RoboDK station: Simulation_roboDK.rdk

Station Simulation_roboDK (saved by RoboDK 5.7.3). Poses are relative to the parent item; angles as X-Y-Z fixed-axis rotations.
  - object Manikin_1 at (0, 0, 0) mm, geometry from Manikin_1.STEP
  - frame Human_Base at (0, 958, 0) mm
    - frame hipL_abduction at (63.26, -78.51, -37.42) mm, rotated rx 0 ry 0 rz -7.94 deg
      - frame hipL_flexion at (0, 0, 0) mm
        - frame hipL_rotation at (0, 0, 0) mm
          - frame kneeL_flexion at (67.44, -393.44, -12.97) mm
            - frame ankleL_flexion at (42.46, -394.54, 0) mm, rotated rx 0 ry 0 rz 7.94 deg
              - item type 7 Manikin_1-pied_g
            - item type 7 Manikin_1-tibia_g
          - item type 7 Manikin_1-cuisse_g
    - frame shoulderL_abduction at (206.4, 423.68, 12.96) mm, rotated rx 0 ry 0 rz -42 deg
      - frame shoulderL_flexion at (0, 0, 0) mm
        - frame shoulderL_rotation at (0, 0, 0) mm
          - frame elbowL_flexion at (155.8, -191.9, 27.9) mm
            - frame wristL_flexion at (148.7, -146.81, 80.89) mm
              - frame wristL_deviation at (0, 0, 0) mm
                - item type 7 Manikin_1-main_g
            - item type 7 Manikin_1-avant_bras_g
          - item type 7 Manikin_1-bras_g
    - frame hipR_abduction at (-70.11, -75.34, -37.06) mm, rotated rx 0 ry 0 rz 10.84 deg
      - frame hipR_flexion at (0, 0, 0) mm
        - frame hipR_rotation at (0, 0, 0) mm
          - frame kneeR_flexion at (-86.5, -385.51, -37.91) mm
            - frame ankleR_flexion at (-60.5, -382.31, -26.03) mm, rotated rx 0 ry 0 rz -10.84 deg
              - item type 7 Manikin_1-pied_d_1
              - item type 7 Manikin_1-pied_d_2
            - item type 7 Manikin_1-tibia_d_1
            - item type 7 Manikin_1-tibia_d_2
          - item type 7 Manikin_1-cuisse_d
    - frame shoulderR_abduction at (-136.98, 400.49, -20) mm, rotated rx 0 ry 0 rz -63.21 deg
      - frame shoulderR_flexion at (0, 0, 0) mm, rotated rx 57.65 ry 0 rz 0 deg
        - frame shoulderR_rotation at (0, 0, 0) mm, rotated rx 0 ry 29.61 rz 0 deg
          - frame elbowR_flexion at (-80.76, -228.86, 52.14) mm, rotated rx -95.28 ry 0 rz 0 deg
            - frame forearmR_rotation at (0, 0, 0) mm, rotated rx 0 ry 25.7 rz 0 deg
              - frame wristR_flexion at (-76.34, -195.54, 87.27) mm, rotated rx -9.18 ry 0 rz 0 deg
                - frame wristR_deviation at (0, 0, 0) mm, rotated rx 0 ry 0 rz 5.97 deg
                  - item type 7 Manikin_1-main_d
              - item type 7 Manikin_1-avant_bras_d
          - item type 7 Manikin_1-bras_d
    - item type 7 Manikin_1-bassin
    - item type 7 Manikin_1-tete
    - item type 7 Manikin_1-torso
  - Python program fix_segments (listed below)
  - object Table at (0, 900, 485) mm, size 1100 x 900 x 550 mm
  - object Piece at (80, 940, 300) mm, size 80 x 80 x 80 mm
  - Python program play_trajectory_robodk (listed below)
  - Python program Position_0 (listed below)

--- Python program fix_segments ---
# -*- coding: utf-8 -*-
"""
fix_reattache_segments.py — Repare le mannequin eclate a la reouverture du
.rdk SANS rebuild (quelques secondes), en re-jouant le re-basage geometrique
perdu a la sauvegarde.

Cause (diagnostic du 10/06) : pour les sous-solides type 7 (courbes issues
du Split), le .rdk sauve les points BRUTS d'origine — la compensation posee
par setParentStatic au moment du rig n'est PAS persistee. A l'ouverture,
RoboDK applique la transformation du frame parent sur ces points bruts
-> double transformation -> mannequin eclate. Les frames, vrais items a
pose persistee, restent corrects.

Remede, segment par segment :
  1) memoriser la pose relative de chaque frame, puis remettre chaque
     frame en etat de CONSTRUCTION (translation seule, rotation identite —
     l'etat dans lequel le rig d'origine a pose ses compensations)
  2) setParent(station)      — detache en KEEP-RELATIVE : la compensation
     (identite au chargement) ne change pas -> le segment retombe sur ses
     points bruts = position d'import, mannequin recompose
     setParentStatic(frame)  — re-attache en preservant l'absolu : la
     compensation F_build^-1 est re-posee, exactement comme au rig
  3) restaurer les poses memorisees (garde-a-vous, jambes resserrees) :
     la geometrie suit les frames

!! NE PAS envelopper dans RDK.Render(False) : le re-basage des type 7
echoue silencieusement sans rendu actif (constate le 10/06 — deux
tentatives identiques en Render(False) = aucun effet, la meme sequence
render actif fonctionne).

A relancer A CHAQUE OUVERTURE du .rdk (la sauvegarde re-perd le re-basage).
Filet de securite si etat incoherent : scripts/rebuild_operateur.py (~30 s).

!! PAS IDEMPOTENT : sur une station SAINE (fraichement rebuildee ou deja
reparee), le re-basage s'appliquerait une fois de trop et eclaterait le
mannequin. Une garde detecte l'etat via un segment du tronc et refuse de
tourner si la station est saine (--force pour outrepasser).

Usage (RoboDK ouvert, station chargee) :
    python fix_reattache_segments.py [--skip nom1,nom2] [--force]
    --skip  : segments a ne pas toucher (ex. deja repares a la main)
    --force : sauter la garde de detection
"""
import math
import sys
import time
from pathlib import Path
sys.path.insert(0, str(Path(__file__).resolve().parent))
from robolink import Robolink, ITEM_TYPE_FRAME
from robodk.robomath import transl

# ancres d'import des segments du tronc (cf. build_human_robodk.ANCHORS),
# en dur pour que le script reste autonome une fois embarque dans la station
TRONC = {"tete": (20, 1584, 30), "torso": (15, 1260, 0), "bassin": (0, 958, 0)}

skip = set()
if "--skip" in sys.argv:
    skip = set(sys.argv[sys.argv.index("--skip") + 1].split(","))

t0 = time.time()
RDK = Robolink()
station = RDK.ActiveStation()
print("Station :", station.Name())


def _d(a, b):
    return math.sqrt(sum((x - y) ** 2 for x, y in zip(a, b)))


def garde_station_cassee():
    """True si le mannequin est eclate (double transformation detectee)."""
    for it in RDK.ItemList():
        if it.Type() != 7:
            continue
        part = it.Name().split("-", 1)[-1]
        if part not in TRONC:
            continue
        bb = it.setParam("BoundingBox")
        c = [(bb["min"][i] + bb["max"][i]) / 2.0 for i in range(3)]
        a = TRONC[part]
        F = it.Parent().PoseAbs().rows
        fa = [sum(F[i][j] * a[j] for j in range(3)) + F[i][3] for i in range(3)]
        d_sain, d_casse = _d(c, a), _d(c, fa)
        etat = "CASSEE (double transformation)" if d_casse < d_sain else "saine"
        print(f"Garde ({part}) : d_sain={d_sain:.0f} mm, d_casse={d_casse:.0f} mm -> station {etat}")
        return d_casse < d_sain
    sys.exit("Garde impossible : aucun segment du tronc (tete/torso/bassin) trouve.")


if "--force" not in sys.argv and not garde_station_cassee():
    sys.exit("Rien a faire — relancer avec --force pour outrepasser la garde.")

frames = RDK.ItemList(ITEM_TYPE_FRAME)
solids = [it for it in RDK.ItemList() if it.Type() == 7]
if not solids:
    sys.exit("Rien a reparer : aucun sous-solide type 7 dans la station.")
parent_of = {}
for s in solids:
    nm = s.Name()
    if nm in skip or nm.split("-", 1)[-1] in skip:
        print(f"  (skip : {nm})")
        continue
    p = s.Parent()
    if p.Type() == 3:
        parent_of[s] = p
    else:
        print(f"  (ignore : {nm} n'est pas sous un frame)")
print(f"{len(frames)} frames, {len(parent_of)} segments a re-attacher")

# 1) frames -> etat de construction (translation seule)
saved = []
for fr in frames:
    pose = fr.Pose()
    saved.append((fr, pose))
    r = pose.rows
    fr.setPose(transl(r[0][3], r[1][3], r[2][3]))

# 2) re-basage : detacher en keep-relative, re-attacher en statique
for s, fr in parent_of.items():
    s.setParent(station)
    s.setParentStatic(fr)
    print(f"  re-attache : {s.Name():26s} -> {fr.Name()}")

# 3) restaurer les poses (garde-a-vous, jambes resserrees, ...)
for fr, pose in saved:
    fr.setPose(pose)

print(f"OK — {len(parent_of)} segments re-attaches en {time.time() - t0:.1f} s")

--- Python program play_trajectory_robodk ---
# -*- coding: utf-8 -*-
"""
play_trajectory_robodk.py

Plays back a precomputed 7-DOF joint trajectory (from
src/export_trajectory_for_robodk.py) on a RoboDK mannequin arm -- the
playback half of the PINN/RoboDK digital-twin integration (see chat,
2026-08-10). Deliberately mirrors old/Tache_Bras.py's own structure
(Robolink() + named Frame items + REST pose * local rotation + fixed-rate
render loop) since that's the established, working pattern in this
project for animating this kind of rig -- just without Tache_Bras's IK/
choreography, since here the trajectory is already fully precomputed by
the PINN.

Run this under RoboDK's OWN embedded Python (has robodk/robolink/numpy
already, confirmed 2026-08-10), with the target RoboDK station open:
    C:\\RoboDK\\Python-Embedded\\python.exe play_trajectory_robodk.py <csv_path>

IMPORTANT -- JOINT_MAP below is an unverified best guess and WILL need
your input once the new 7-DOF station exists:
  - rig_frame: must match the exact Frame item name in your new station.
    Left blank (None) for all 7 by default -- fill these in first, the
    script exits immediately listing what it can't find otherwise.
  - axis: which local axis (x/y/z) that frame rotates about. Copied from
    old/config.py's SEGMENTS (the existing 7-DOF chain scaffold in this
    project) as a starting point -- verify against however you actually
    build the new joints, they may not match.
  - sign: +1 or -1. DBAS22's angle convention for a given column is not
    guaranteed to match whichever direction you wire the corresponding
    RoboDK axis to rotate. Use --probe (below) to check each joint
    in isolation and flip signs until the motion looks anatomically
    correct, exactly how Tache_Bras.py's original author calibrated
    elbowL_flexion's sign via manual probing (see its "_probe_coude"
    comment) -- there's no way to get this right without the actual rig
    in front of you.

Usage:
    play_trajectory_robodk.py <csv_path>              play back a trajectory
    play_trajectory_robodk.py --probe [step_deg]       one joint at a time,
                                                        +step_deg (default 20)
                                                        from rest, paused for
                                                        visual check between
                                                        each -- run this FIRST
"""
import csv
import math
import sys
from pathlib import Path

from robolink import Robolink, ITEM_TYPE_FRAME
from robodk.robomath import rotx, roty, rotz

# DBAS22 column -> (rig frame name, local axis, sign). Order matches
# dataset.JOINT_COLS (sp, sr, ay, ep, fy, hp, hr); rig frame names/axes
# follow old/config.py's SEGMENTS naming (shoulder_abduction, ...,
# wrist_deviation) as a starting point -- see module docstring.
JOINT_MAP = {
    # Frame names confirmed against the live station (Simulation_roboDK.rdk,
    # 2026-08-10) via robolink -- RIGHT arm, since s1 (the trial used in
    # trajectories/s1_tgt50_*.csv) is right-handed (arm_side='R'). Axes/
    # signs are still the config.py-derived best guess -- run --probe
    # before trusting them.
    "sp": {"rig_frame": "shoulderR_flexion", "axis": "x", "sign": +1},
    "sr": {"rig_frame": "shoulderR_abduction", "axis": "z", "sign": +1},
    "ay": {"rig_frame": "shoulderR_rotation", "axis": "y", "sign": +1},
    "ep": {"rig_frame": "elbowR_flexion", "axis": "x", "sign": +1},
    "fy": {"rig_frame": "forearmR_rotation", "axis": "y", "sign": +1},
    "hp": {"rig_frame": "wristR_flexion", "axis": "x", "sign": +1},
    "hr": {"rig_frame": "wristR_deviation", "axis": "z", "sign": +1},
}
ROT = {"x": rotx, "y": roty, "z": rotz}

DT = 0.04  # s/frame during playback (~25 fps of applied poses; actual
           # wall-clock rate is capped by RoboDK's render time, same
           # caveat Tache_Bras.py notes for its own DT)


def _load_csv(path):
    with open(path, newline="") as f:
        r = csv.reader(f)
        header = next(r)
        rows = [[float(x) for x in row] for row in r]
    cols = {name: i for i, name in enumerate(header)}
    return header, cols, rows


def _get_frames(rdk):
    frames = {}
    missing = []
    for col, spec in JOINT_MAP.items():
        name = spec["rig_frame"]
        if name is None:
            missing.append(f"{col} (rig_frame not set)")
            continue
        fr = rdk.Item(name, ITEM_TYPE_FRAME)
        if not fr.Valid():
            missing.append(f"{col} -> '{name}' (not found in station)")
            continue
        frames[col] = fr
    if missing:
        sys.exit("Fill in / fix JOINT_MAP before running -- problems:\n  "
                  + "\n  ".join(missing))
    return frames


def probe(rdk, step_deg):
    """One joint at a time: rest pose, then rest + step_deg, paused for a
    visual check. Run this first on a new station to calibrate axis/sign
    in JOINT_MAP -- there's no way to get this right without eyeballing
    the actual rig."""
    frames = _get_frames(rdk)
    rest = {col: fr.Pose() for col, fr in frames.items()}

    for col, fr in frames.items():
        axis, sign = JOINT_MAP[col]["axis"], JOINT_MAP[col]["sign"]
        print(f"\n--- probing '{col}' (rig frame '{JOINT_MAP[col]['rig_frame']}', "
              f"axis={axis}, current sign={sign:+d}) ---")
        fr.setPose(rest[col])
        rdk.Render(True)
        input(f"  showing REST. Enter to apply +{step_deg} deg...")
        fr.setPose(rest[col] * ROT[axis](sign * math.radians(step_deg)))
        rdk.Render(True)
        input(f"  applied. Check the motion matches '{col}'s expected anatomical "
              f"direction, then Enter to continue (edit JOINT_MAP's sign if not)...")
        fr.setPose(rest[col])
    rdk.Render(True)
    print("\nProbe done, all joints back at rest.")


def play(rdk, csv_path):
    header, cols, rows = _load_csv(csv_path)
    frames = _get_frames(rdk)
    rest = {col: fr.Pose() for col, fr in frames.items()}
    t_idx = cols["t"]

    print(f"Loaded {len(rows)} frames from {csv_path} "
          f"(duration {rows[-1][t_idx] - rows[0][t_idx]:.2f}s)")

    import time
    t0 = time.time()
    for i, row in enumerate(rows):
        for col, fr in frames.items():
            axis, sign = JOINT_MAP[col]["axis"], JOINT_MAP[col]["sign"]
            angle_deg = sign * row[cols[col]]
            fr.setPose(rest[col] * ROT[axis](math.radians(angle_deg)))
        rdk.Render(True)
        target = t0 + (i + 1) * DT
        remaining = target - time.time()
        if remaining > 0:
            time.sleep(remaining)
    print("Playback done.")


def main():
    rdk = Robolink()
    print("Station:", rdk.ActiveStation().Name())

    if "--probe" in sys.argv:
        idx = sys.argv.index("--probe")
        step = float(sys.argv[idx + 1]) if len(sys.argv) > idx + 1 else 20.0
        probe(rdk, step)
        return

    if len(sys.argv) < 2:
        sys.exit("Usage: play_trajectory_robodk.py <csv_path>  |  --probe [step_deg]")
    play(rdk, Path(sys.argv[1]))


if __name__ == "__main__":
    main()

--- Python program Position_0 ---
# -*- coding: utf-8 -*-
"""
Position_0.py — Remet le mannequin au GARDE-A-VOUS exact (position zero).

A lancer quand on veut repartir d'un etat propre : apres une animation
interrompue, un script qui a laisse le bras en l'air, ou des residus
accumules (chaque animation se termine a quelques degres pres ; les petits
ecarts s'additionnent au fil des runs).

Reconstruit le zero du rig (cf. rig_active_station.py, section 8) :
  - les 22 DDL -> rotation IDENTITE (la translation du repere ne bouge
    jamais, on la conserve telle quelle) ;
  - epaule du cote X+ (= gauche) : rotz(-42 deg) pour plaquer le bras que
    la pose STEP d'origine ecarte du corps ;
  - jambes resserrees : cheville ramenee a l'aplomb de la hanche (angle
    recalcule depuis les positions des reperes, pied contre-tourne).

Ne touche ni la Table, ni la Piece, ni la camera.
    C:\\RoboDK\\Python-Embedded\\python.exe scripts\\Position_0.py
"""
import math
import sys
from robolink import Robolink, ITEM_TYPE_FRAME
from robodk.robomath import Mat, rotz

DOF = [
    "shoulderL_abduction", "shoulderL_flexion", "shoulderL_rotation",
    "elbowL_flexion", "wristL_flexion", "wristL_deviation",
    "shoulderR_abduction", "shoulderR_flexion", "shoulderR_rotation",
    "elbowR_flexion", "forearmR_rotation", "wristR_flexion", "wristR_deviation",
    # forearmR_rotation added 2026-08-10: the new 7th-DOF joint inserted
    # between elbowR_flexion and wristR_flexion (right arm only) for the
    # PINN digital-twin work -- this original 22-DOF list predates that
    # change and never reset it, so any leftover rotation on that one
    # frame from a prior script run survives every "reset to zero" call,
    # which can visually detach the forearm/hand from the rest of the
    # body depending on how those meshes are parented to it.
    "hipL_abduction", "hipL_flexion", "hipL_rotation", "kneeL_flexion",
    "ankleL_flexion",
    "hipR_abduction", "hipR_flexion", "hipR_rotation", "kneeR_flexion",
    "ankleR_flexion",
]


def _zero(fr):
    """Rotation identite, translation conservee."""
    p = fr.Pose()
    fr.setPose(Mat([[1, 0, 0, p[0, 3]], [0, 1, 0, p[1, 3]],
                    [0, 0, 1, p[2, 3]], [0, 0, 0, 1]]))


def remettre_a_zero(RDK, verbose=True):
    """Remet les 22 DDL au garde-a-vous exact. Importable par les scripts
    d'animation (a appeler AVANT de capturer le repos)."""
    F = {}
    for nm in DOF:
        fr = RDK.Item(nm, ITEM_TYPE_FRAME)
        if not fr.Valid():
            sys.exit(f"ERREUR : repere {nm} introuvable — rig 22 DDL absent ?")
        F[nm] = fr

    # 1) tout a zero (les positions absolues redeviennent celles de la pose STEP)
    for nm in DOF:
        _zero(F[nm])

    # 2) bras gauche (cote X+) plaque le long du corps
    F["shoulderL_abduction"].setPose(
        F["shoulderL_abduction"].Pose() * rotz(math.radians(-42.0)))

    # 3) jambes resserrees : meme calcul que le rig (cheville a l'aplomb de la
    #    hanche), possible car a l'etape 1 les reperes sont aux positions STEP
    for u in ("R", "L"):
        hp = F[f"hip{u}_abduction"].PoseAbs()
        ap = F[f"ankle{u}_flexion"].PoseAbs()
        ang = math.atan2(ap[0, 3] - hp[0, 3], hp[1, 3] - ap[1, 3])
        F[f"hip{u}_abduction"].setPose(F[f"hip{u}_abduction"].Pose() * rotz(-ang))
        F[f"ankle{u}_flexion"].setPose(F[f"ankle{u}_flexion"].Pose() * rotz(ang))
        if verbose:
            print(f"  jambes resserrees ({u}) : {math.degrees(ang):+.1f} deg")


if __name__ == "__main__":
    RDK = Robolink()
    print("Station :", RDK.ActiveStation().Name())
    remettre_a_zero(RDK)
    RDK.Render(True)
    print("Position 0 : mannequin au garde-a-vous.")
